// TIA Portal V19 export
TYPE "LEXCHANGETRAY_typeConstraintWorkstationEm_toConstraintRollerRecieve"
// stored: Access Published
   STRUCT
      feedback { S7_SetPoint := 'True'} : "LEXCHANGETRAY_typeConstraintRollerEm_toConstraintWorkstationFeedback";
      req { S7_SetPoint := 'True'} : "LEXCHANGETRAY_typeConstraintRollerEm_toConstraintWorkstationReq";
   END_STRUCT;
END_TYPE
